Staubli VAL3: encodeAck.pgx

public program encodeAck(RosSimpleMsg& x_msg)
begin
  // Copyright (c) 2016, Ocado Technology - Robotics Research Team
  // Copyright (c) 2021, Institute for Factory Automation and Production Systems (FAPS)
  //
  // Licensed under the Apache License, Version 2.0 (the "License");
  // you may not use this file except in compliance with the License.
  // You may obtain a copy of the License at
  //
  //     http://www.apache.org/licenses/LICENSE-2.0
  //
  // Unless required by applicable law or agreed to in writing, software
  // distributed under the License is distributed on an "AS IS" BASIS,
  // WITHOUT WARRANTIES OR CONDITIONS OF ANY KIND, either express or implied.
  // See the License for the specific language governing permissions and
  // limitations under the License.



  switch x_msg.header.nMsgType

    case SimpleMsg:MsgType.JOINT_TRAJ_PT
      call encTrajPtAck()
    break

    case SimpleMsg:MsgType.JOINT_TRAJ_PT_F
      call encTrajPtFAck()
    break

    // Staubli specific
    case Staubli:MsgType.SET_DRIVE_POWER
      call Staubli:encSetDrvPwrAck()
    break

    case Staubli:MsgType.WRITE_SINGLE_IO
      call Staubli:encWriSingIOAck()
    break

    case Staubli:MsgType.VELOCITY_CFG
      call Staubli:encodeVelCfgAck()
    break

    case Staubli:MsgType.VELOCITY_CMD
      call Staubli:encodeVelCmdAck()
    break

    default
      //region @DEBUG
      if (bDebugMode and nDebugLevel<=5)
        call printDebug("encodeAck: switch (msgType)",true)
        call printDebug("ERROR: unknown msg type",false)
      endIf
      //endregion
    break
  endSwitch
end
